TYPE MNG_DataArray : ARRAY[1..MNG_BUFFER_SIZE] OF DWORD; (* user data of max. length *)
END_TYPE

(* stored: Version 1.1.0.1, ProductVersion 3.1.0.25
   DUT MNG_DataArray: Id {a5523c87-2ee0-4fe3-b2d2-b83dfe582647} *)
